// TwinCAT 3 PLC project SchmittTriggerTests
// ProgramVersion: 3.1.4026.22
// libraries:
//   Tc2_Standard, * (Beckhoff Automation GmbH)
//   Tc2_System, * (Beckhoff Automation GmbH)
//   TcUnit, * (www.tcunit.org)
//   T1SchmittTrigger_Plc,newest,Tc3 Project
// project tree:
//   / PlcTask.TcTTO
//   POUs/ FB_SchmittTriggerConsumer.TcPOU, MAIN.TcPOU
// real-time tasks:
//   TASK PlcTask: cycle T#10ms, priority 20, ADS port 350

CONFIGURATION SchmittTriggerTests
    RESOURCE PLC ON TwinCAT3
        TASK PlcTask(INTERVAL := T#10ms, PRIORITY := 21);
        PROGRAM MAIN WITH PlcTask : MAIN;
    END_RESOURCE
END_CONFIGURATION

// ---- POUs/MAIN.TcPOU
PROGRAM MAIN
VAR
END_VAR

END_PROGRAM

// ---- POUs/FB_SchmittTriggerConsumer.TcPOU
FUNCTION_BLOCK FB_SchmittTriggerConsumer
VAR
    trigger : T1SchmittTrigger_Plc.FB_SchmittTrigger;
    bLastState : BOOL;
END_VAR

trigger(fInput := 0.5);
bLastState := trigger.Step();

END_FUNCTION_BLOCK
